REGION Network 45: Enable HMI Code View
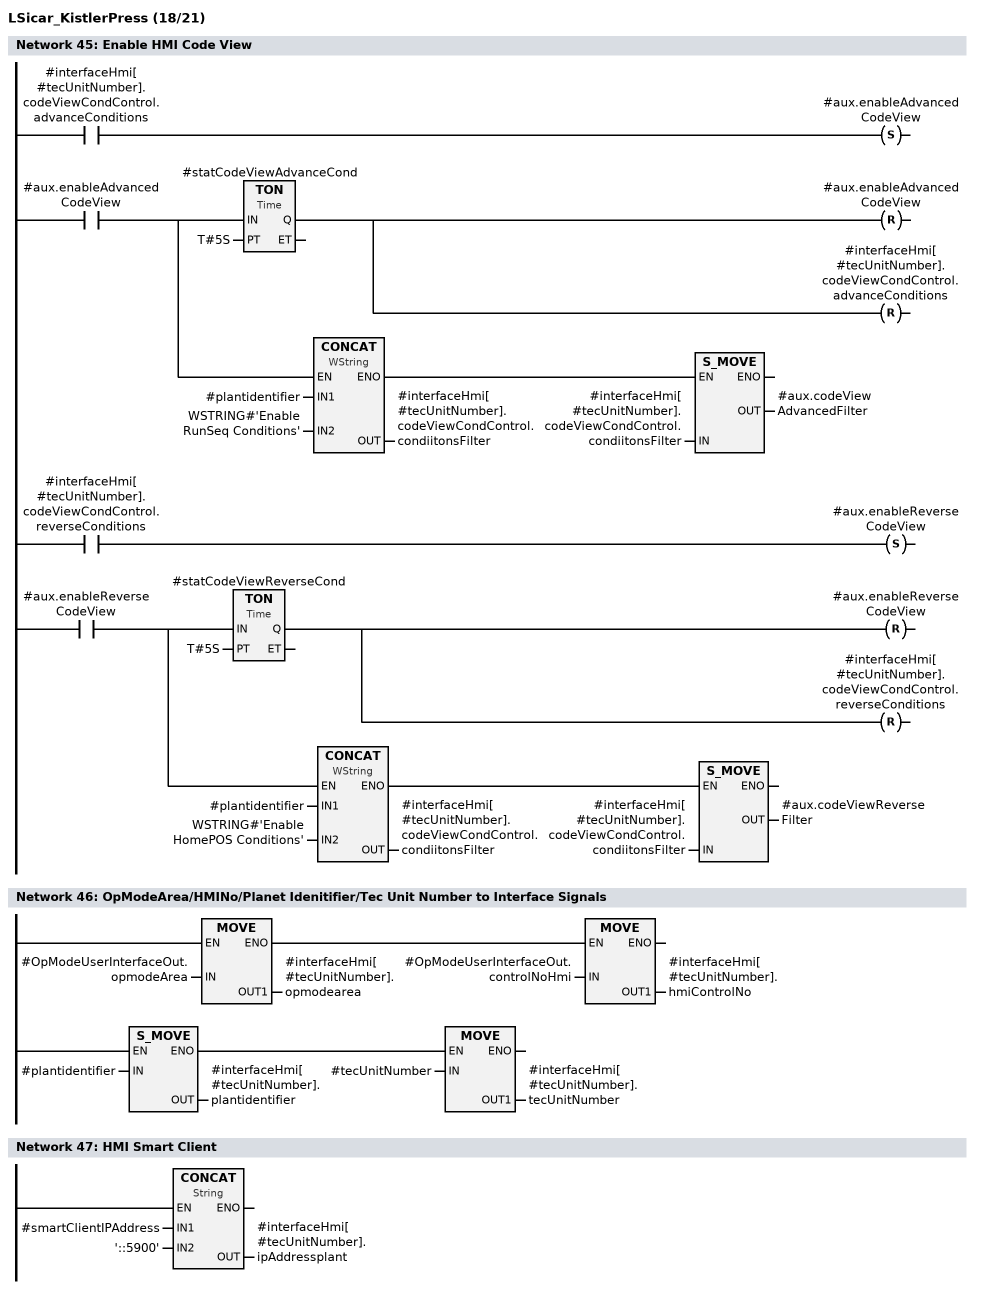
   RUNG wire#powerrail
      Contact( #interfaceHmi[#tecUnitNumber].codeViewCondControl.advanceConditions )
      S_Coil( #aux.enableAdvancedCodeView )
   END_RUNG
   RUNG wire#powerrail
      Contact( #aux.enableAdvancedCodeView )
      wire#w1
      { S7_Templates := "time_type := Time" } #statCodeViewAdvanceCond.TON(pt := T#5S, et =>)
      wire#w2
      R_Coil( #aux.enableAdvancedCodeView )
   END_RUNG
   RUNG wire#w2
      R_Coil( #interfaceHmi[#tecUnitNumber].codeViewCondControl.advanceConditions )
   END_RUNG
   RUNG wire#w1
      { S7_Templates := "[card := 2, str_type := WString]" } CONCAT(IN1 := #plantidentifier, IN2 := WSTRING#'Enable RunSeq Conditions', OUT => #interfaceHmi[#tecUnitNumber].codeViewCondControl.condiitonsFilter)
      S_Move(in := #interfaceHmi[#tecUnitNumber].codeViewCondControl.condiitonsFilter, out => #aux.codeViewAdvancedFilter)
   END_RUNG
   RUNG wire#powerrail
      Contact( #interfaceHmi[#tecUnitNumber].codeViewCondControl.reverseConditions )
      S_Coil( #aux.enableReverseCodeView )
   END_RUNG
   RUNG wire#powerrail
      Contact( #aux.enableReverseCodeView )
      wire#w3
      { S7_Templates := "time_type := Time" } #statCodeViewReverseCond.TON(pt := T#5S, et =>)
      wire#w4
      R_Coil( #aux.enableReverseCodeView )
   END_RUNG
   RUNG wire#w4
      R_Coil( #interfaceHmi[#tecUnitNumber].codeViewCondControl.reverseConditions )
   END_RUNG
   RUNG wire#w3
      { S7_Templates := "[card := 2, str_type := WString]" } CONCAT(IN1 := #plantidentifier, IN2 := WSTRING#'Enable HomePOS Conditions', OUT => #interfaceHmi[#tecUnitNumber].codeViewCondControl.condiitonsFilter)
      S_Move(in := #interfaceHmi[#tecUnitNumber].codeViewCondControl.condiitonsFilter, out => #aux.codeViewReverseFilter)
   END_RUNG
   // the same network as SCL:
   IF #interfaceHmi[#tecUnitNumber].codeViewCondControl.advanceConditions THEN
       #aux.enableAdvancedCodeView := TRUE;
   END_IF;
   #statCodeViewAdvanceCond(IN := #aux.enableAdvancedCodeView, PT := T#5S);   // TON
   #_w1 := #aux.enableAdvancedCodeView;
   IF #statCodeViewAdvanceCond.Q THEN
       #aux.enableAdvancedCodeView := FALSE;
       #interfaceHmi[#tecUnitNumber].codeViewCondControl.advanceConditions := FALSE;
   END_IF;
   CONCAT(EN := #_w1,
          IN1 := #plantidentifier,
          IN2 := WSTRING#'Enable RunSeq Conditions',
          OUT => #interfaceHmi[#tecUnitNumber].codeViewCondControl.condiitonsFilter,
          ENO => #_w2);
   IF #_w2 THEN
       #aux.codeViewAdvancedFilter := #interfaceHmi[#tecUnitNumber].codeViewCondControl.condiitonsFilter;
   END_IF;
   IF #interfaceHmi[#tecUnitNumber].codeViewCondControl.reverseConditions THEN
       #aux.enableReverseCodeView := TRUE;
   END_IF;
   #statCodeViewReverseCond(IN := #aux.enableReverseCodeView, PT := T#5S);   // TON
   #_w3 := #aux.enableReverseCodeView;
   IF #statCodeViewReverseCond.Q THEN
       #aux.enableReverseCodeView := FALSE;
       #interfaceHmi[#tecUnitNumber].codeViewCondControl.reverseConditions := FALSE;
   END_IF;
   CONCAT(EN := #_w3,
          IN1 := #plantidentifier,
          IN2 := WSTRING#'Enable HomePOS Conditions',
          OUT => #interfaceHmi[#tecUnitNumber].codeViewCondControl.condiitonsFilter,
          ENO => #_w4);
   IF #_w4 THEN
       #aux.codeViewReverseFilter := #interfaceHmi[#tecUnitNumber].codeViewCondControl.condiitonsFilter;
   END_IF;
END_REGION

REGION Network 46: OpModeArea/HMINo/Planet Idenitifier/Tec Unit Number to Interface Signals
   RUNG wire#powerrail
      Move(in := #OpModeUserInterfaceOut.opmodeArea, out1 => #interfaceHmi[#tecUnitNumber].opmodearea)
      Move(in := #OpModeUserInterfaceOut.controlNoHmi, out1 => #interfaceHmi[#tecUnitNumber].hmiControlNo)
   END_RUNG
   RUNG wire#powerrail
      S_Move(in := #plantidentifier, out => #interfaceHmi[#tecUnitNumber].plantidentifier)
      Move(in := #tecUnitNumber, out1 => #interfaceHmi[#tecUnitNumber].tecUnitNumber)
   END_RUNG
   // the same network as SCL:
   #interfaceHmi[#tecUnitNumber].opmodearea := #OpModeUserInterfaceOut.opmodeArea;
   #interfaceHmi[#tecUnitNumber].hmiControlNo := #OpModeUserInterfaceOut.controlNoHmi;
   #interfaceHmi[#tecUnitNumber].plantidentifier := #plantidentifier;
   #interfaceHmi[#tecUnitNumber].tecUnitNumber := #tecUnitNumber;
END_REGION

REGION Network 47: HMI Smart Client
   RUNG wire#powerrail
      { S7_Templates := "[card := 2, str_type := String]" } CONCAT(IN1 := #smartClientIPAddress, IN2 := '::5900', OUT => #interfaceHmi[#tecUnitNumber].ipAddressplant)
   END_RUNG
   // the same network as SCL:
   CONCAT(IN1 := #smartClientIPAddress, IN2 := '::5900', OUT => #interfaceHmi[#tecUnitNumber].ipAddressplant);
END_REGION

REGION Network 48: Map FIx Receieved Data to HMI
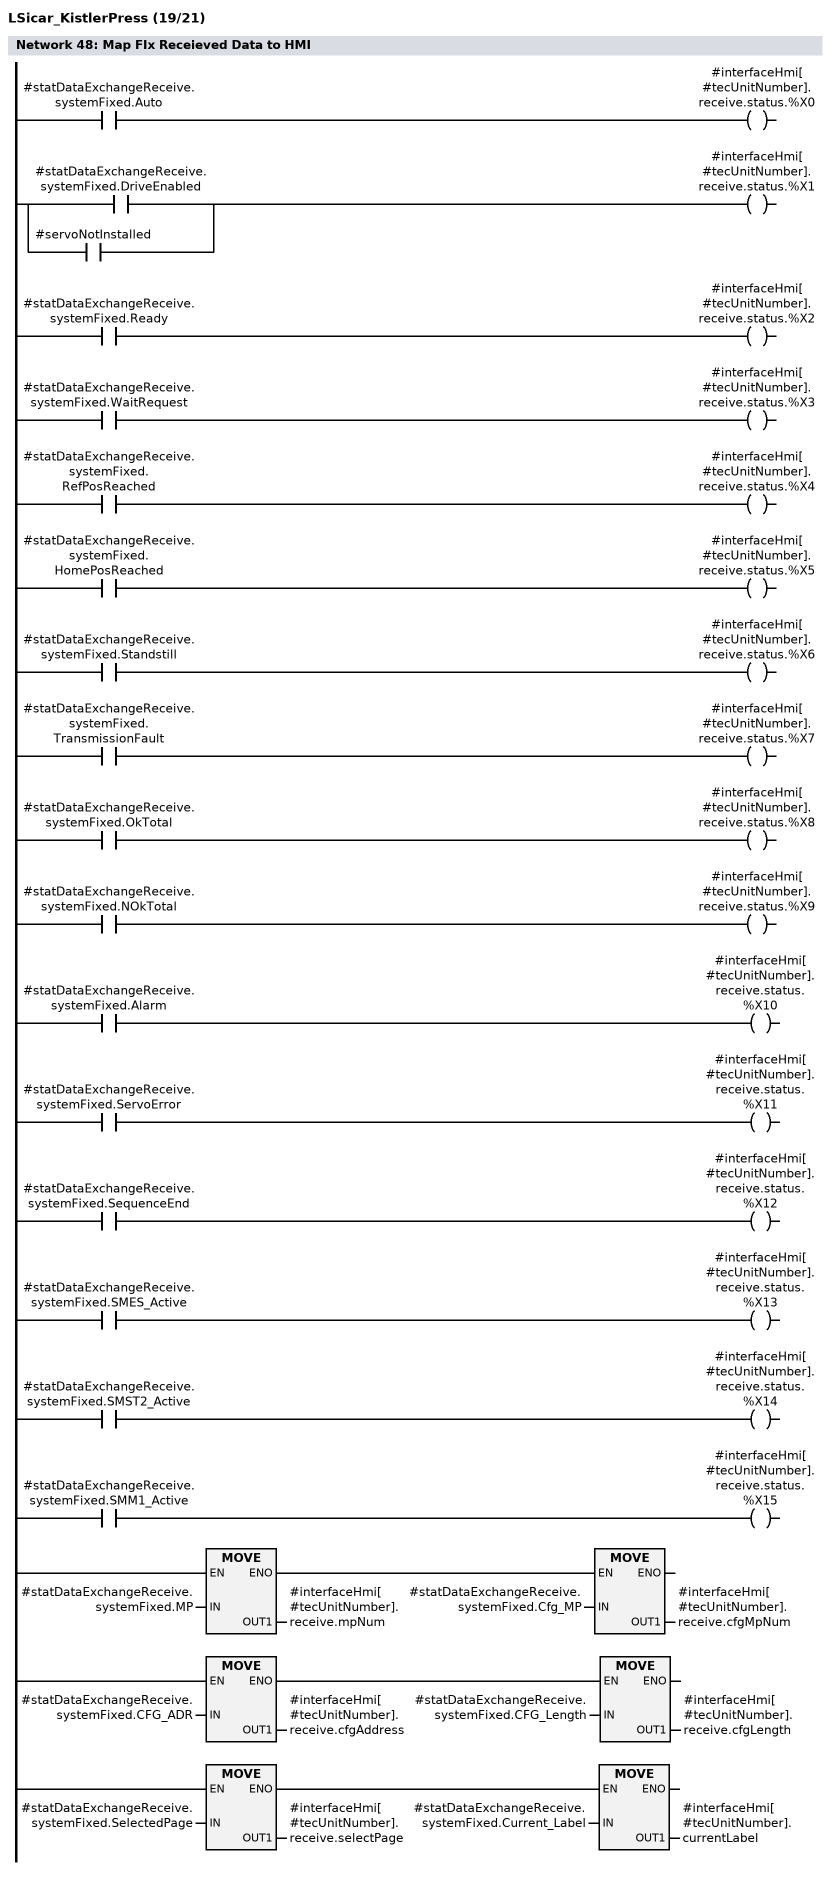
   RUNG wire#powerrail
      Contact( #statDataExchangeReceive.systemFixed.Auto )
      Coil( #interfaceHmi[#tecUnitNumber].receive.status.%X0 )
   END_RUNG
   RUNG wire#powerrail
      Contact( #statDataExchangeReceive.systemFixed.DriveEnabled )
      wire#w1
      Coil( #interfaceHmi[#tecUnitNumber].receive.status.%X1 )
   END_RUNG
   RUNG wire#powerrail
      Contact( #servoNotInstalled )
   END_RUNG wire#w1
   RUNG wire#powerrail
      Contact( #statDataExchangeReceive.systemFixed.Ready )
      Coil( #interfaceHmi[#tecUnitNumber].receive.status.%X2 )
   END_RUNG
   RUNG wire#powerrail
      Contact( #statDataExchangeReceive.systemFixed.WaitRequest )
      Coil( #interfaceHmi[#tecUnitNumber].receive.status.%X3 )
   END_RUNG
   RUNG wire#powerrail
      Contact( #statDataExchangeReceive.systemFixed.RefPosReached )
      Coil( #interfaceHmi[#tecUnitNumber].receive.status.%X4 )
   END_RUNG
   RUNG wire#powerrail
      Contact( #statDataExchangeReceive.systemFixed.HomePosReached )
      Coil( #interfaceHmi[#tecUnitNumber].receive.status.%X5 )
   END_RUNG
   RUNG wire#powerrail
      Contact( #statDataExchangeReceive.systemFixed.Standstill )
      Coil( #interfaceHmi[#tecUnitNumber].receive.status.%X6 )
   END_RUNG
   RUNG wire#powerrail
      Contact( #statDataExchangeReceive.systemFixed.TransmissionFault )
      Coil( #interfaceHmi[#tecUnitNumber].receive.status.%X7 )
   END_RUNG
   RUNG wire#powerrail
      Contact( #statDataExchangeReceive.systemFixed.OkTotal )
      Coil( #interfaceHmi[#tecUnitNumber].receive.status.%X8 )
   END_RUNG
   RUNG wire#powerrail
      Contact( #statDataExchangeReceive.systemFixed.NOkTotal )
      Coil( #interfaceHmi[#tecUnitNumber].receive.status.%X9 )
   END_RUNG
   RUNG wire#powerrail
      Contact( #statDataExchangeReceive.systemFixed.Alarm )
      Coil( #interfaceHmi[#tecUnitNumber].receive.status.%X10 )
   END_RUNG
   RUNG wire#powerrail
      Contact( #statDataExchangeReceive.systemFixed.ServoError )
      Coil( #interfaceHmi[#tecUnitNumber].receive.status.%X11 )
   END_RUNG
   RUNG wire#powerrail
      Contact( #statDataExchangeReceive.systemFixed.SequenceEnd )
      Coil( #interfaceHmi[#tecUnitNumber].receive.status.%X12 )
   END_RUNG
   RUNG wire#powerrail
      Contact( #statDataExchangeReceive.systemFixed.SMES_Active )
      Coil( #interfaceHmi[#tecUnitNumber].receive.status.%X13 )
   END_RUNG
   RUNG wire#powerrail
      Contact( #statDataExchangeReceive.systemFixed.SMST2_Active )
      Coil( #interfaceHmi[#tecUnitNumber].receive.status.%X14 )
   END_RUNG
   RUNG wire#powerrail
      Contact( #statDataExchangeReceive.systemFixed.SMM1_Active )
      Coil( #interfaceHmi[#tecUnitNumber].receive.status.%X15 )
   END_RUNG
   RUNG wire#powerrail
      Move(in := #statDataExchangeReceive.systemFixed.MP, out1 => #interfaceHmi[#tecUnitNumber].receive.mpNum)
      Move(in := #statDataExchangeReceive.systemFixed.Cfg_MP, out1 => #interfaceHmi[#tecUnitNumber].receive.cfgMpNum)
   END_RUNG
   RUNG wire#powerrail
      Move(in := #statDataExchangeReceive.systemFixed.CFG_ADR, out1 => #interfaceHmi[#tecUnitNumber].receive.cfgAddress)
      Move(in := #statDataExchangeReceive.systemFixed.CFG_Length, out1 => #interfaceHmi[#tecUnitNumber].receive.cfgLength)
   END_RUNG
   RUNG wire#powerrail
      Move(in := #statDataExchangeReceive.systemFixed.SelectedPage, out1 => #interfaceHmi[#tecUnitNumber].receive.selectPage)
      Move(in := #statDataExchangeReceive.systemFixed.Current_Label, out1 => #interfaceHmi[#tecUnitNumber].currentLabel)
   END_RUNG
   // the same network as SCL:
   #interfaceHmi[#tecUnitNumber].receive.status.%X0 := #statDataExchangeReceive.systemFixed.Auto;
   #interfaceHmi[#tecUnitNumber].receive.status.%X1 := #statDataExchangeReceive.systemFixed.DriveEnabled OR #servoNotInstalled;
   #interfaceHmi[#tecUnitNumber].receive.status.%X2 := #statDataExchangeReceive.systemFixed.Ready;
   #interfaceHmi[#tecUnitNumber].receive.status.%X3 := #statDataExchangeReceive.systemFixed.WaitRequest;
   #interfaceHmi[#tecUnitNumber].receive.status.%X4 := #statDataExchangeReceive.systemFixed.RefPosReached;
   #interfaceHmi[#tecUnitNumber].receive.status.%X5 := #statDataExchangeReceive.systemFixed.HomePosReached;
   #interfaceHmi[#tecUnitNumber].receive.status.%X6 := #statDataExchangeReceive.systemFixed.Standstill;
   #interfaceHmi[#tecUnitNumber].receive.status.%X7 := #statDataExchangeReceive.systemFixed.TransmissionFault;
   #interfaceHmi[#tecUnitNumber].receive.status.%X8 := #statDataExchangeReceive.systemFixed.OkTotal;
   #interfaceHmi[#tecUnitNumber].receive.status.%X9 := #statDataExchangeReceive.systemFixed.NOkTotal;
   #interfaceHmi[#tecUnitNumber].receive.status.%X10 := #statDataExchangeReceive.systemFixed.Alarm;
   #interfaceHmi[#tecUnitNumber].receive.status.%X11 := #statDataExchangeReceive.systemFixed.ServoError;
   #interfaceHmi[#tecUnitNumber].receive.status.%X12 := #statDataExchangeReceive.systemFixed.SequenceEnd;
   #interfaceHmi[#tecUnitNumber].receive.status.%X13 := #statDataExchangeReceive.systemFixed.SMES_Active;
   #interfaceHmi[#tecUnitNumber].receive.status.%X14 := #statDataExchangeReceive.systemFixed.SMST2_Active;
   #interfaceHmi[#tecUnitNumber].receive.status.%X15 := #statDataExchangeReceive.systemFixed.SMM1_Active;
   #interfaceHmi[#tecUnitNumber].receive.mpNum := #statDataExchangeReceive.systemFixed.MP;
   #interfaceHmi[#tecUnitNumber].receive.cfgMpNum := #statDataExchangeReceive.systemFixed.Cfg_MP;
   #interfaceHmi[#tecUnitNumber].receive.cfgAddress := #statDataExchangeReceive.systemFixed.CFG_ADR;
   #interfaceHmi[#tecUnitNumber].receive.cfgLength := #statDataExchangeReceive.systemFixed.CFG_Length;
   #interfaceHmi[#tecUnitNumber].receive.selectPage := #statDataExchangeReceive.systemFixed.SelectedPage;
   #interfaceHmi[#tecUnitNumber].currentLabel := #statDataExchangeReceive.systemFixed.Current_Label;
END_REGION

REGION Network 49: Map Fix Send Data to HMI
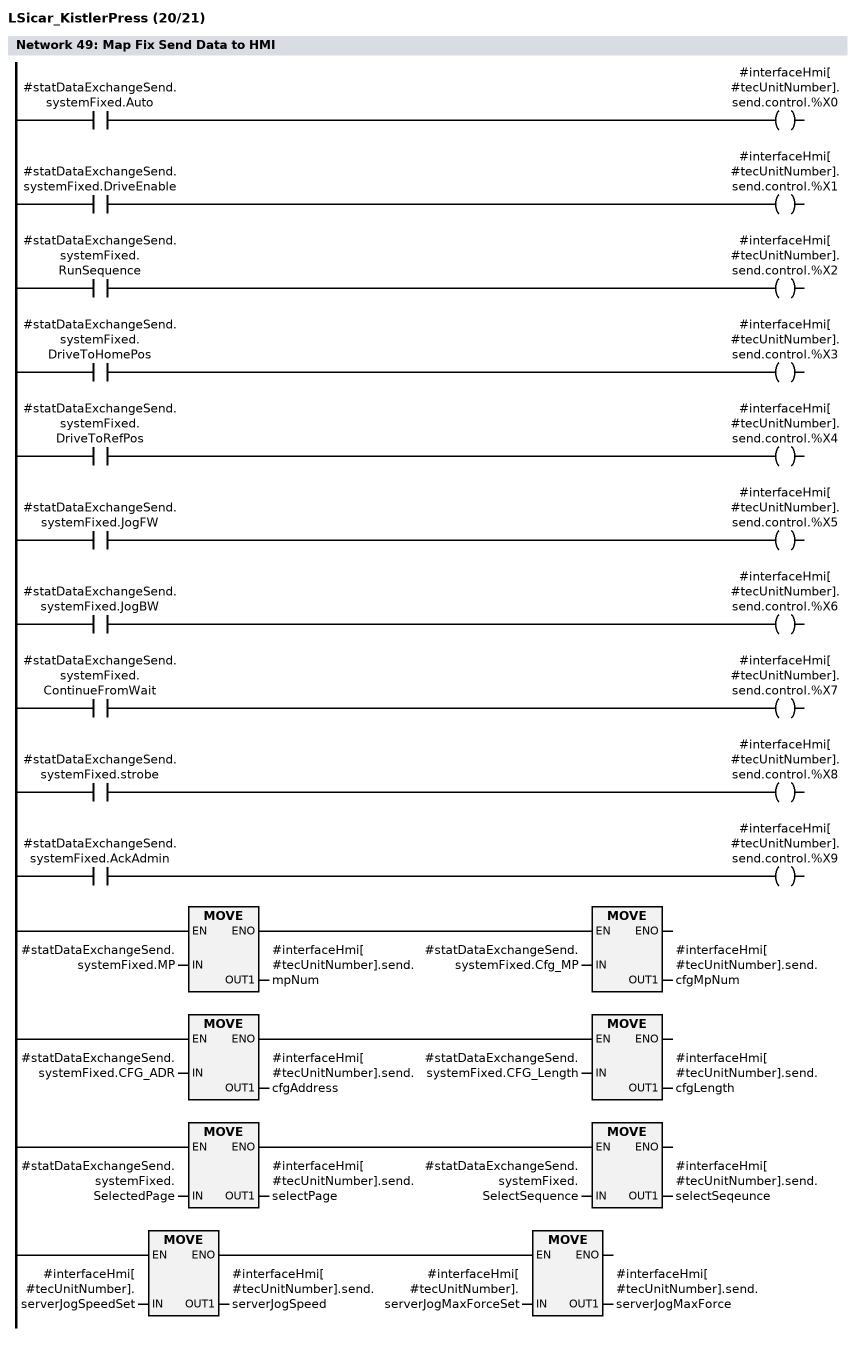
   RUNG wire#powerrail
      Contact( #statDataExchangeSend.systemFixed.Auto )
      Coil( #interfaceHmi[#tecUnitNumber].send.control.%X0 )
   END_RUNG
   RUNG wire#powerrail
      Contact( #statDataExchangeSend.systemFixed.DriveEnable )
      Coil( #interfaceHmi[#tecUnitNumber].send.control.%X1 )
   END_RUNG
   RUNG wire#powerrail
      Contact( #statDataExchangeSend.systemFixed.RunSequence )
      Coil( #interfaceHmi[#tecUnitNumber].send.control.%X2 )
   END_RUNG
   RUNG wire#powerrail
      Contact( #statDataExchangeSend.systemFixed.DriveToHomePos )
      Coil( #interfaceHmi[#tecUnitNumber].send.control.%X3 )
   END_RUNG
   RUNG wire#powerrail
      Contact( #statDataExchangeSend.systemFixed.DriveToRefPos )
      Coil( #interfaceHmi[#tecUnitNumber].send.control.%X4 )
   END_RUNG
   RUNG wire#powerrail
      Contact( #statDataExchangeSend.systemFixed.JogFW )
      Coil( #interfaceHmi[#tecUnitNumber].send.control.%X5 )
   END_RUNG
   RUNG wire#powerrail
      Contact( #statDataExchangeSend.systemFixed.JogBW )
      Coil( #interfaceHmi[#tecUnitNumber].send.control.%X6 )
   END_RUNG
   RUNG wire#powerrail
      Contact( #statDataExchangeSend.systemFixed.ContinueFromWait )
      Coil( #interfaceHmi[#tecUnitNumber].send.control.%X7 )
   END_RUNG
   RUNG wire#powerrail
      Contact( #statDataExchangeSend.systemFixed.strobe )
      Coil( #interfaceHmi[#tecUnitNumber].send.control.%X8 )
   END_RUNG
   RUNG wire#powerrail
      Contact( #statDataExchangeSend.systemFixed.AckAdmin )
      Coil( #interfaceHmi[#tecUnitNumber].send.control.%X9 )
   END_RUNG
   RUNG wire#powerrail
      Move(in := #statDataExchangeSend.systemFixed.MP, out1 => #interfaceHmi[#tecUnitNumber].send.mpNum)
      Move(in := #statDataExchangeSend.systemFixed.Cfg_MP, out1 => #interfaceHmi[#tecUnitNumber].send.cfgMpNum)
   END_RUNG
   RUNG wire#powerrail
      Move(in := #statDataExchangeSend.systemFixed.CFG_ADR, out1 => #interfaceHmi[#tecUnitNumber].send.cfgAddress)
      Move(in := #statDataExchangeSend.systemFixed.CFG_Length, out1 => #interfaceHmi[#tecUnitNumber].send.cfgLength)
   END_RUNG
   RUNG wire#powerrail
      Move(in := #statDataExchangeSend.systemFixed.SelectedPage, out1 => #interfaceHmi[#tecUnitNumber].send.selectPage)
      Move(in := #statDataExchangeSend.systemFixed.SelectSequence, out1 => #interfaceHmi[#tecUnitNumber].send.selectSeqeunce)
   END_RUNG
   RUNG wire#powerrail
      Move(in := #interfaceHmi[#tecUnitNumber].serverJogSpeedSet, out1 => #interfaceHmi[#tecUnitNumber].send.serverJogSpeed)
      Move(in := #interfaceHmi[#tecUnitNumber].serverJogMaxForceSet, out1 => #interfaceHmi[#tecUnitNumber].send.serverJogMaxForce)
   END_RUNG
   // the same network as SCL:
   #interfaceHmi[#tecUnitNumber].send.control.%X0 := #statDataExchangeSend.systemFixed.Auto;
   #interfaceHmi[#tecUnitNumber].send.control.%X1 := #statDataExchangeSend.systemFixed.DriveEnable;
   #interfaceHmi[#tecUnitNumber].send.control.%X2 := #statDataExchangeSend.systemFixed.RunSequence;
   #interfaceHmi[#tecUnitNumber].send.control.%X3 := #statDataExchangeSend.systemFixed.DriveToHomePos;
   #interfaceHmi[#tecUnitNumber].send.control.%X4 := #statDataExchangeSend.systemFixed.DriveToRefPos;
   #interfaceHmi[#tecUnitNumber].send.control.%X5 := #statDataExchangeSend.systemFixed.JogFW;
   #interfaceHmi[#tecUnitNumber].send.control.%X6 := #statDataExchangeSend.systemFixed.JogBW;
   #interfaceHmi[#tecUnitNumber].send.control.%X7 := #statDataExchangeSend.systemFixed.ContinueFromWait;
   #interfaceHmi[#tecUnitNumber].send.control.%X8 := #statDataExchangeSend.systemFixed.strobe;
   #interfaceHmi[#tecUnitNumber].send.control.%X9 := #statDataExchangeSend.systemFixed.AckAdmin;
   #interfaceHmi[#tecUnitNumber].send.mpNum := #statDataExchangeSend.systemFixed.MP;
   #interfaceHmi[#tecUnitNumber].send.cfgMpNum := #statDataExchangeSend.systemFixed.Cfg_MP;
   #interfaceHmi[#tecUnitNumber].send.cfgAddress := #statDataExchangeSend.systemFixed.CFG_ADR;
   #interfaceHmi[#tecUnitNumber].send.cfgLength := #statDataExchangeSend.systemFixed.CFG_Length;
   #interfaceHmi[#tecUnitNumber].send.selectPage := #statDataExchangeSend.systemFixed.SelectedPage;
   #interfaceHmi[#tecUnitNumber].send.selectSeqeunce := #statDataExchangeSend.systemFixed.SelectSequence;
   #interfaceHmi[#tecUnitNumber].send.serverJogSpeed := #interfaceHmi[#tecUnitNumber].serverJogSpeedSet;
   #interfaceHmi[#tecUnitNumber].send.serverJogMaxForce := #interfaceHmi[#tecUnitNumber].serverJogMaxForceSet;
END_REGION

REGION Network 50: Generate Alarm for Pro Diag
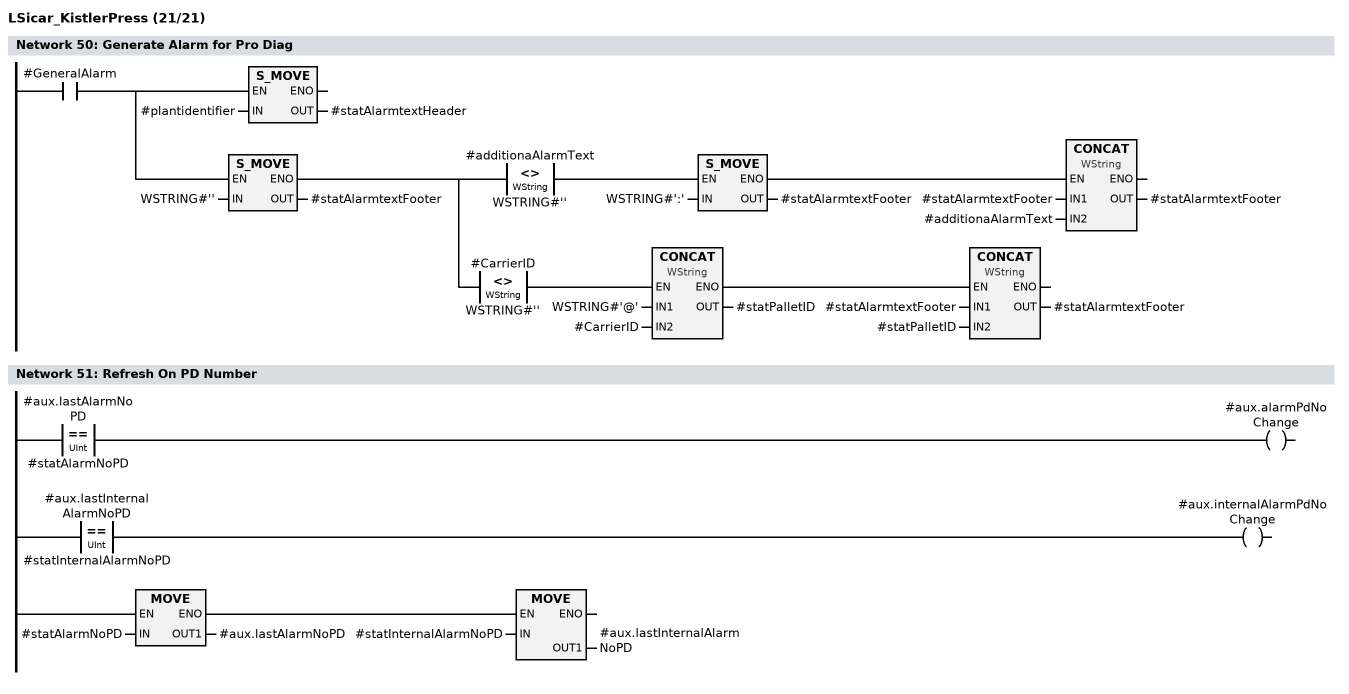
   RUNG wire#powerrail
      Contact( #GeneralAlarm )
      wire#w1
      S_Move(in := #plantidentifier, out => #statAlarmtextHeader)
   END_RUNG
   RUNG wire#w1
      S_Move(in := WSTRING#'', out => #statAlarmtextFooter)
      wire#w2
      { S7_Templates := "SrcType := WString" } NE_Contact(in1 := #additionaAlarmText, in2 := WSTRING#'')
      S_Move(in := WSTRING#':', out => #statAlarmtextFooter)
      { S7_Templates := "[card := 2, str_type := WString]" } CONCAT(IN1 := #statAlarmtextFooter, IN2 := #additionaAlarmText, OUT => #statAlarmtextFooter)
   END_RUNG
   RUNG wire#w2
      { S7_Templates := "SrcType := WString" } NE_Contact(in1 := #CarrierID, in2 := WSTRING#'')
      { S7_Templates := "[card := 2, str_type := WString]" } CONCAT(IN1 := WSTRING#'@', IN2 := #CarrierID, OUT => #statPalletID)
      { S7_Templates := "[card := 2, str_type := WString]" } CONCAT(IN1 := #statAlarmtextFooter, IN2 := #statPalletID, OUT => #statAlarmtextFooter)
   END_RUNG
   // the same network as SCL:
   IF #GeneralAlarm THEN
       #statAlarmtextHeader := #plantidentifier;
       #statAlarmtextFooter := WSTRING#'';
   END_IF;
   IF #GeneralAlarm AND (#additionaAlarmText <> WSTRING#'') THEN
       #statAlarmtextFooter := WSTRING#':';
       CONCAT(IN1 := #statAlarmtextFooter, IN2 := #additionaAlarmText, OUT => #statAlarmtextFooter);
   END_IF;
   CONCAT(EN := #GeneralAlarm AND (#CarrierID <> WSTRING#''),
          IN1 := WSTRING#'@',
          IN2 := #CarrierID,
          OUT => #statPalletID,
          ENO => #_w1);
   IF #_w1 THEN
       CONCAT(IN1 := #statAlarmtextFooter, IN2 := #statPalletID, OUT => #statAlarmtextFooter);
   END_IF;
END_REGION

REGION Network 51: Refresh On PD Number
   RUNG wire#powerrail
      { S7_Templates := "SrcType := UInt" } EQ_Contact(in1 := #aux.lastAlarmNoPD, in2 := #statAlarmNoPD)
      Coil( #aux.alarmPdNoChange )
   END_RUNG
   RUNG wire#powerrail
      { S7_Templates := "SrcType := UInt" } EQ_Contact(in1 := #aux.lastInternalAlarmNoPD, in2 := #statInternalAlarmNoPD)
      Coil( #aux.internalAlarmPdNoChange )
   END_RUNG
   RUNG wire#powerrail
      Move(in := #statAlarmNoPD, out1 => #aux.lastAlarmNoPD)
      Move(in := #statInternalAlarmNoPD, out1 => #aux.lastInternalAlarmNoPD)
   END_RUNG
   // the same network as SCL:
   #aux.alarmPdNoChange := #aux.lastAlarmNoPD = #statAlarmNoPD;
   #aux.internalAlarmPdNoChange := #aux.lastInternalAlarmNoPD = #statInternalAlarmNoPD;
   #aux.lastAlarmNoPD := #statAlarmNoPD;
   #aux.lastInternalAlarmNoPD := #statInternalAlarmNoPD;
END_REGION
END_FUNCTION_BLOCK
